Fanuc KAREL source: PROG_LIST.kl

PROGRAM T
%NOLOCKGROUP
VAR
 v0 : STRING[40]
 v1 : INTEGER
 v2 : INTEGER
 v3 : INTEGER
 v4 : ARRAY[10] OF STRING[40]
 v5 : INTEGER
 v6 : INTEGER
 v7 : INTEGER
BEGIN
 PROG_LIST(v0, v1, v2, v3, v4, v5, v6, v7)
END T
